FUNCTION_BLOCK FB_Component_SingleValve IMPLEMENTS I_Component
VAR_INPUT
// Interface vars
	sName			: STRING[20];
	bEnable     	: BOOL;
	//eMode       	: E_ComponentMode;
END_VAR

VAR_IN_OUT
	bOutput			: BOOL;
END_VAR

VAR_OUTPUT
	// interface vars
	eState			: E_ComponentState;
	iErrorCode		: INT;
	sStatusText 	: STRING[50];
END_VAR

METHOD M_Extend : BOOL
VAR_INPUT
END_VAR
IF bEnable AND eState = E_ComponentState.READY THEN
	bOutput := TRUE;	
END_IF;
END_METHOD

METHOD M_Halt : BOOL
bOutput := FALSE;
eState := E_ComponentState.HALTED;
END_METHOD

METHOD M_Retract : BOOL
VAR_INPUT
END_VAR
IF bEnable AND eState = E_ComponentState.READY THEN
	bOutput := FALSE;
END_IF;
END_METHOD

{warning 'add method implementation '}
METHOD M_Start : BOOL
IF eState <> E_ComponentState.BUSY THEN
	eState := E_ComponentState.READY;
END_IF;
END_METHOD

{warning 'add method implementation '}
METHOD M_Stop : BOOL
IF eState <> E_ComponentState.BUSY THEN
	eState := E_ComponentState.DONE;
END_IF
END_METHOD

END_FUNCTION_BLOCK

(* stored: Version 1.1.0.1, ProductVersion 3.1.4024.15
   POU FB_Component_SingleValve: Id {e241cca9-8ad1-4d32-953d-80e7ad832e70}, SpecialFunc None
   Method M_Extend: Id {116184ed-7298-4777-808a-4e90b7472e93}
   Method M_Halt: Id {d6d164e4-6ff2-4655-bb53-7508a90ca844}
   Method M_Retract: Id {32527918-9b92-4347-97af-cfb47d794b1c}
   Method M_Start: Id {3b5e4edb-f27f-4280-94ac-c799f1f4bcbc}
   Method M_Stop: Id {8f25114a-9d10-4e85-92e5-9d523c21fcd3} *)
